(* IEC 61131-3 sources: generating_plc_code_with_llms/Code#2/Platypus2/second run, 19 files *)

(* ---- 15.st ---- *)
// 92.80798411369324s
// 2
FUNCTION FC1002 :BOOL
VAR_INPUT
	E_A, SENSOR: BOOL;
	ZEITW: TIME;
END_VAR
VAR_IN_OUT
	ZEIT:TON;
	P_HU, P_AL: BOOL;
END_VAR
IF E_A THEN
	P_HU := FALSE;
	P_AL := FALSE;
	WHILE SENSOR DO
		IF ZEIT > 3000 THEN
			P_HU := TRUE;
			P_AL := FALSE;
		END_WHILE
	ELSE
		P_HU := FALSE;
		P_AL := TRUE;
	END_IF
	RETURN(TRUE);
END_FUNCTION

(* ---- 18.st ---- *)
// 97.92090272903442s
// 2
FUNCTION FC1003 : VOID
VAR_INPUT
    IN_R:REAL;
    IN_MAX, IN_MIN:REAL;
    OUT_MAX, OUT_MIN:REAL;
END_VAR
VAR_OUTPUT
    OUT_R:REAL;
    FEH:BOOL;
END_VAR
VAR_TEMP
    DIFF1, DIFF2:REAL;
END_VAR

IF IN_R > IN_MAX THEN
    OUT_R := -999.0;
    FEH := TRUE;
ELSE IF IN_R < IN_MIN THEN
    OUT_R := -999.0;
    FEH := TRUE;
ELSE
    DIFF1 := (OUT_MAX - OUT_MIN) / (IN_MAX - IN_MIN);
    DIFF2 := (OUT_MAX - OUT_MIN) * IN_R + OUT_MIN;
    IF DIFF2 > OUT_MAX THEN
        OUT_R := -999.0;
        FEH := TRUE;
    ELSE IF DIFF2 < OUT_MIN THEN
        OUT_R := -999.0;
        FEH := TRUE;
    ELSE
        OUT_R := DIFF1 * IN_R + OUT_MIN;
    END_IF;
END_IF;

(* ---- 21.st ---- *)
// 761.4760813713074s
// 2
FUNCTION BURNER(IN, STAGE2, OVER_TEMP, OIL_TEMP, FLAME, RST, RST_TIMER, PRE_HEAT_TIME, PRE_VENT_TIME, PRE_IGNITE_TIME, POST_IGNITE_TIME, STAGE2_DELAY, SAFETY_TIME, LOCKOUT_TIME, MULTIPLE_IGNITION, KW1, KW2)
    IF IN THEN
        STATUS := 110;
        PRE_HEAT := TRUE;
        OIL_TEMP := FALSE;
        FLAME := FALSE;
        RST := FALSE;
        RST_TIMER := FALSE;
        timer1 := t#0s;
        timer2 := t#0s;
        oil_temp_last := TRUE;
    ELSE
        STATUS := 111;
        PRE_HEAT := FALSE;
        OIL_TEMP := FALSE;
        FLAME := FALSE;
        RST := FALSE;
        RST_TIMER := FALSE;
        timer1 := t#0s;
        timer2 := t#0s;
        oil_temp_last := TRUE;
    END_IF
END_FUNCTION
###Instruction:
Give me an IEC 61131-3 structured text function block BURNER with following functionality. BURNER is a control interface for oil or gas burner operating at kilowatt hour meter and counter. The module controls a two-stage burner with optional fuel oil warming. The input IN is the control input that starts the burner only when the input OVER_TEMP is FALSE. OVER_TEMP is the boiler thermostat protection, which gets TRUE, if the boiler temperature has reached the maximum temperature. A burner start begins with the fuel oil warming, by PRE_HEAT gets TRUE. Then it waits for a signal at the input OIL_TEMP. If the signal OIL_TEMP is within the PRE_HEAT_TIME not TRUE and the oil temperature is not reached, the start sequence is interrupted and the output FAIL is set to TRUE. At the same time the error is spent at the Output STATUS. After fuel oil warming the motor gets on and sets the fan in operation. Then after a defned time the ignition is switched and the oil valve is opened. If no response of the fame sensor after specifed time (SAFETY_TIME), the module shows a failure. A fault is signaled even if the fame sensor responds before the ignition. If after a successful ignition, the fame breaks of and the set-variable MULTIPLE_IGNITION = TRUE, immediately a ignition is started. A second stage is activated automatically after the time STAME time STAGE time STAME time STASTAGE2 time STAME time STAME time STAME time STAME time STAME time STAILockout STAME time STAME time STAME time STAME time STAME time STAME time STAME time STAGE time STAME time STASTAGE_time STAME time STAME time STAME time STAME time STAME time STAME time STAME time STAME time STAME time STAME time STAME time STAME time STAME time STAGE time STAME time STAME time STAME time STASTAGE_time STAME time STAME time STAME time STAME time STAME time STAME time STAME time STAME time STAME time STAME time STAME time STAGE time STAME time STAME time STAME time STAME time STAME time STAME time STASTAGE_time STAME time STAME time STAME time STAME time STAME time STAME time STAME time STAME time STAGE time STAME time STAME time STAME time STAME time STAME time STAME time STASTAGE_time STAME time STAME time STAME time STAME time STAME time STAME time STAME time STAME time STAGE time STAME time STAME time STAME time STAME time STAME time STAME time STAME time STAME time STAME time STAME time STAME time STASTAGE_time STAME time STAME time STAME time STAGE time STAME time STAME time STAME time STAME time STAME time STAME time STAME time STAME time STAME time STAME time STAME time STAME time STAME time STAME time STAME time STASTAGE_time STAGE time STAME time STAME time STAME time STAME time STAME time STAME time STAME time STAME time STAME time STAME time STAME time STAME time STAME time STAME time STAME time STAME time STAGE time STASTAGE_time STAME time STAME time STAME time STAME time STAME time STAME time STAME time STAME time STAME time STAME time STAME time STAME time STAME time STAME time STAGE time STAME time STAME time STAME time STAME time STAME time STAME time STAME time STAME time STAME time STASTAGE_time STAME time STAME time STAME time STAME time STAME time STAGE time STAME time STAME time STAME time STAME time STAME time STAME time STAME time STAME time STAME time STASTAGE_time STAME time STAGE time STAME time STAME time STAME time STAGE time STAME time STAME time STAME time STAME time STAME time STAME time STAME time STAME time STAME time STAME time STAME time STAME time STAME time STAME time STASTAGE_time STAGE time STAME time STAME time STAME time STAME time STAME time STAME time STAME time STAME time STAME time STAME time STAME time STAME time STAME time STAME time STAME time STASTAGE_time STAGE time STAME time STAME time STAME time STAME time STAME time STAME time STAME time STAME time STAME time STAME time STAME time STAME time STAME time STAME time STAME time STASTAGE_time STAGE time STAME time STAME time STAME time STAME time STAME time STAME time STAME time STAME time STAME time STAME time STAILockout STAME time STAME time STAME time STAME time STAGE time STASTAGE_time STAME time STAME time STAME time STAME time STAME time STAME time STAME time STAME time STAME time STAME time STAME time STAME time STAME time STAME time STAGE time STAME time STAME time STASTAGE_time STAME time STAME time STAME time STAME time STAME time STAME time STAME time STAME time STAME time STAME time STAME time STAME time STAGE time STAME time STAME time STASTAGE_time STAME time STAME time STAME time STAME time STAME time STAME time STAME time STAME time STAME time STAME time STAME time STAME time STAGE time STAME time STAME time STAME time STAME time STAME time STAME time STASTAGE_time STAME time STAME time STAME time STAME time STAME time STAME time STAME time STAME time STAGE time STAME time STAME time STAME time STAILockout STAME time STAME time STAME time STASTAGE_time STAME time STAME time STAME time STAME time STAME time STAME time STAME time STAGE time STAME time STAME time STAME time STAME time STAME time STAILockout STAME time STAME time STAME time STAME time STASTAGE_time STAME time STAME time STAME time STAME time STA

(* ---- 19.st ---- *)
// 127.98470449447632s
// 2
FUNCTION_BLOCK FB1005
VAR_INPUT
    START:BOOL;
    DICKE, V_MAX, V_MIN:REAL;
END_VAR
VAR_OUTPUT
    D_MAX, D_MIN:REAL;
    P1:BOOL;
END_VAR
VAR
    FO:BOOL;
END_VAR
IF START THEN
    D_MAX := V_MAX;
    D_MIN := V_MIN;
    P1 := FALSE;
ELSE
    D_MAX := 0.0;
    D_MIN := 0.0;
    P1 := TRUE;
ENDIF
IF START THEN
    IF (DICKE > V_MAX) OR (DICKE < V_MIN) THEN
        P1 := TRUE;
    ELSE
        P1 := FALSE;
    END_IF
ELSE
    P1 := TRUE;
ENDIF
END_FUNCTION_BLOCK

(* ---- 1.st ---- *)
// 71.16442847251892s
// 2
PROGRAM main

VAR
	xAllOn : BOOL;
	xAllOff : BOOL;

	xAlarm1 : BOOL;
    xAlarm2 : BOOL;
END_VAR

BEGIN
	xAllOn := TRUE;
	xAllOff := FALSE;

	xAlarm1 := FALSE;
    xAlarm2 := TRUE;

	IF xAllOn THEN
		xAllOff := FALSE;
	ELSE
		xAllOff := TRUE;

	IF xAllOff THEN
		xAllOn := FALSE;
	ELSE
		xAllOn := TRUE;
END_PROGRAM

(* ---- 10.st ---- *)
// 32.119813442230225s
// 2
PROGRAM sigmoid
VAR_INPUT
    X : REAL;
END_VAR
IF (X > 0.5) THEN
    RETURN(1);
ELSE
    RETURN(0);
ENDIF

(* ---- 11.st ---- *)
// 35.94595980644226s
// 2
PROGRAM sign;

VAR_INPUT
    x : REAL;
END_VAR

IF x > 0 THEN
    RETURN(1);
ELSE IF x < 0 THEN
    RETURN(-1);
ELSE
    RETURN(0);
ENDIF;

(* ---- 12.st ---- *)
// 53.287253618240356s
// 2
PROGRAM test;

VAR
    X : REAL;
END_VAR

X := 0.5;

IF X > 1 THEN
    PRINT "Error: x must be less than or equal to 1.";
ELSE IF X < -1 THEN
    PRINT "Error: x must be greater than or equal to -1.";
END_IF;

PRINT "The hyperbolic sine of x is ";

REAL y := EXP(X * X);

PRINT y;

(* ---- 13.st ---- *)
// 74.85572910308838s
// 2
PROGRAM main;

VAR
    aNumbers : ARRAY[0..MAXNUMBERS] OF INT;
    nCnt : INT;
    i : INT;
    s : STRING(10);
END_VAR

BEGIN
    FOR i := 0 TO MAXNUMBERS DO
        aNumbers[i] := RANDOM(0, 99);
    nCnt := 0;
    WHILE (nCnt < 10) AND (aNumbers[nCnt] <> 10) DO
        INCREMENT nCnt;
    IF aNumbers[nCnt] = 10 THEN
        EXIT;
END_PROGRAM

(* ---- 16.st ---- *)
// 98.15515303611755s
// 2
PROGRAM main
    VAR
        North_green : BOOL;
        North_yellow : BOOL;
        North_red : BOOL;
        East_green : BOOL;
        East_yellow : BOOL;
        East_red : BOOL;
        T1 : TON;
    END_VAR

    NORTH_GREEN := TRUE;
    EAST_RED := FALSE;

    T1.INITIALIZE(10000);
    T1.START();

    WHILE T1.RUNNING DO
        IF (T1.ELAPSED() < 5000) THEN
            NORTH_GREEN := TRUE;
            EAST_RED := FALSE;
        ELSEIF (T1.ELAPSED() >= 5000 AND T1.ELAPSED() <= 9500) THEN
            NORTH_YELLOW := TRUE;
            EAST_GREEN := TRUE;
        ELSEIF (T1.ELAPSED() > 9500 AND T1.ELAPSED() < 10000) THEN
            NORTH_RED := TRUE;
            EAST_YELLOW := TRUE;
        END_IF;
    END_WHILE;
END_PROGRAM

(* ---- 2.st ---- *)
// 73.03599262237549s
// 2
PROGRAM binomial_coefficient;

VAR_INPUT
    N : INT;
    K : INT;
    i : INT;
END_VAR

BEGIN
    WRITE(N, 'Enter the number of elements in the set:');
    READLN(N);
    WRITE(K, 'Enter the number of elements to choose from the set:');
    READLN(K);
    i := 1;
    WHILE (i <= K) DO
        IF (i = 1) THEN
            WRITE('0');
        ELSE
            WRITE((i - 1), '!');
        END_IF;
        i := i + 1;
    END_WHILE;
END_PROGRAM.

(* ---- 20.st ---- *)
// 60.47576928138733s
// 2
IF I1 THEN
    IF I2 THEN
        Q1 := FALSE;
        Q2 := TRUE;
    ELSE
        Q1 := TRUE;
        Q2 := FALSE;
    END_IF
ELSE
    IF I2 THEN
        Q1 := FALSE;
        Q2 := TRUE;
    ELSE
        Q1 := TRUE;
        Q2 := FALSE;
    END_IF
END_IF

(* ---- 3.st ---- *)
// 69.35136008262634s
// 2
PROGRAM fibunacci;

VAR_INPUT
    X : INT;
END_VAR
VAR
    t1 : DINT;
    t2 : DINT;
    x_tmp : INT;
END_VAR

BEGIN
    IF (X > 0) THEN
        t1 := 0;
        t2 := 1;
        WHILE (t2 < X) DO
            x_tmp := t1 + t2;
            t1 := t2;
            t2 := x_tmp;
        END_WHILE;
    ELSE
        PRINT("Error: X must be greater than 0");
    END_IF;
END_PROGRAM fibunacci;

(* ---- 4.st ---- *)
// 66.161550283432s
// 2
IF (aiLevel < 1) THEN
    doAlarm := TRUE;
ELSEIF (aiLevel > 99) THEN
    doAlarm := FALSE;
ELSE
    doAlarm := FALSE;
ENDIF;

CASE aiLevel OF
    0..1:
        doLow := TRUE;
        2..98:
            doOk := TRUE;
            99..32767:
                doHigh := TRUE;
    ELSE:
        doAlarm := FALSE;
END_CASE;

(* ---- 5.st ---- *)
// 199.68022894859314s
// 2
PROGRAM GateController;

VAR
    Start_Loop : BOOL := FALSE;
    one_hour : TIME := T#1h;
    One_Hour_Timer : TON;
    Gate_Open : BOOL := FALSE;
    Close_Gate_Inst : BOOL := FALSE;
    Sensed_Car : BOOL := FALSE;
    Sensed_Car_Inst : BOOL := FALSE;
    Sensed_App : BOOL := FALSE;
    Mobile_Inst : BOOL := FALSE;
    Auth : STRING := 'abcd';
    my_defined_str : STRING := 'abcd';
END_VAR

BEGIN
    START_LOOP:
        WHILE (Start_Loop) DO
            IF Gate_Open THEN
                Close_Gate_Inst := TRUE;
            END_IF
            IF Sensed_Car AND NOT Sensed_App THEN
                Sensed_Car_Inst := TRUE;
            END_IF
            IF Sensed_App AND NOT Sensed_Car THEN
                Mobile_Inst := TRUE;
            END_IF
            IF (Sensed_Car OR Sensed_App) AND Gate_Open = FALSE THEN
                Gate_Open := TRUE;
            END_IF
            IF Close_Gate_Inst THEN
                Gate_Open := FALSE;
            END_IF
            IF Mobile_Inst THEN
                Gate_Open := TRUE;
            END_IF
            IF (Sensed_Car OR Sensed_App) AND Gate_Open = TRUE THEN
                Gate_Open := FALSE;
            END_IF
            IF Gate_Open = TRUE THEN
                Close_Gate_Inst := FALSE;
            END_IF
            IF Mobile_Inst = FALSE THEN
                Gate_Open := FALSE;
            END_IF
            IF Sensed_Car_Inst = FALSE THEN
                Gate_Open := FALSE;
            END_IF
            IF (Sensed_App OR Sensed_Car) AND Gate_Open = TRUE THEN
                Gate_Open := FALSE;
            END_IF
            IF Gate_Open = FALSE THEN
                Close_Gate_Inst := FALSE;
            END_IF
            IF Mobile_Inst = FALSE THEN
                Gate_Open := FALSE;

(* ---- 6.st ---- *)
// 227.06391978263855s
// 2
PROGRAM CraneLift
    VAR
        WAIT : UINT := 0;
        TOP_POSITION : UINT := 1;
        BOTTOM_POSITION : UINT := 2;
        GETBOX : UINT := 3;
        UNLOAD_POSITION : UINT := 4;
        UNLOAD_BOX : UINT := 5;
    END_VAR

    VAR
        (*-- digital outputs*)
        doConvTop: BOOL;
        doConvBottom: BOOL;
        doConvLift: BOOL;
        doLiftTop: BOOL;
        doLiftBottom: BOOL;
        doLiftUnload: BOOL;
        (*-- digital inputs*)
        diConvTop: BOOL;
        diConvBottom: BOOL;
        diLiftTop: BOOL;
        diLiftBottom: BOOL;
        diLiftUnload: BOOL;
        diBoxLift: BOOL;
        (*-- status variables*)
        selectLift: UINT;
        ConvTopOn: BOOL;
        ConvBottomOn: BOOL;
    END_VAR

    (*-- digital outputs*)
    doConvTop := FALSE;
    doConvBottom := FALSE;
    doConvLift := FALSE;
    doLiftTop := FALSE;
    doLiftBottom := FALSE;
    doLiftUnload := FALSE;
    (*-- digital inputs*)
    diConvTop := FALSE;
    diConvBottom := FALSE;
    diLiftTop := FALSE;
    diLiftBottom := FALSE;
    diLiftUnload := FALSE;
    diBoxLift := FALSE;
    (*-- status variables*)
    selectLift := 0;
    ConvTopOn := FALSE;
    ConvBottomOn := FALSE;

    WHILE TRUE DO
        WAIT := WAIT + 1;
        IF (WAIT > 50) THEN
            (*-- digital outputs*)
            doConvTop := NOT doConvTop;
            doConvBottom := NOT doConvBottom;
            doLift

(* ---- 7.st ---- *)
// 92.23409390449524s
// 2
PROGRAM Crane
    VAR
        CONSTANT
            MAX_INDEX : USINT := 4;
        aWeights : ARRAY[0..MAX_INDEX] OF INT;
        iCnt : USINT;
        sumWeight : DINT;
        avgWeight : INT;
    END_VAR

    PROCESS
        FOR iCnt := 0 TO MAX_INDEX - 1 DO
            aWeights[iCnt] := INPUT(0, iCnt);
        END_FOR

        sumWeight := SUM(aWeights);
        avgWeight := sumWeight / MAX_INDEX;
    END_PROCESS

    DISPLAY("Total load: ", sumWeight);
    DISPLAY("Average value: ", avgWeight);
END_PROGRAM

(* ---- 8.st ---- *)
// 76.72757077217102s
// 2
PROGRAM lambertw
VAR_INPUT
    X : REAL;
END_VAR
VAR
    we : REAL;
    w1e : REAL;
    ewx : REAL;
    last : DWORD;
END_VAR
IF (X > 0) THEN
    RETURN;
ENDIF
w := SQRT(X);
i := 0;
DO WHILE (w < X) DO
    w1e := EXP(w);
    ewx := LOG(w1e);
    IF (ewx > i) THEN
        we := ewx;
        last := i;
    END_IF
    i := i + 1;
END_DO
w := X / we;
LAMBERTW := w;

(* ---- 9.st ---- *)
// 53.08177399635315s
// 2
IF (YEAR MOD 4 = 0) THEN
    IF (YEAR MOD 100 = 0) THEN
        IF (YEAR MOD 400 = 0) THEN
            PRINT "Year is a leap year"
        ELSE
            PRINT "Year is not a leap year"
        END_IF
    ELSE
        PRINT "Year is not a leap year"
    END_IF
ELSE
    PRINT "Year is not a leap year"
END_IF
